{attribute 'GeneratedUsingTerminal: EL6688-0000-0016'}
{attribute addProperty BoxType "EL6688-0000-0016"}
{attribute addProperty Id "SYNC_InputsAT %I*SYNC_Inputs_971453DD4WcStateAT %I*WcState_9091E0EB2InfoDataAT %I*InfoData_1088C70510"}
{attribute addProperty CRC "79085063"}
{attribute addProperty Size "16"}
TYPE EL6688_04B6BE07 EXTENDS EtcSlaveTerminalBase_947E5A46 :
STRUCT
	{attribute addProperty Name "SYNC_Inputs"}
	SYNC_Inputs : SYNC_Inputs_971453DD;
	{attribute addProperty Name "WcState"}
	WcState : WcState_9091E0EB;
	{attribute addProperty Name "InfoData"}
	InfoData : InfoData_1088C705;
END_STRUCT
END_TYPE

(* stored: Version 1.2.0.0, ProductVersion 3.1.4024.9
   DUT EL6688_04B6BE07: Id {151d9ded-ef58-41cf-97fc-c6e3c3fa7438} *)
